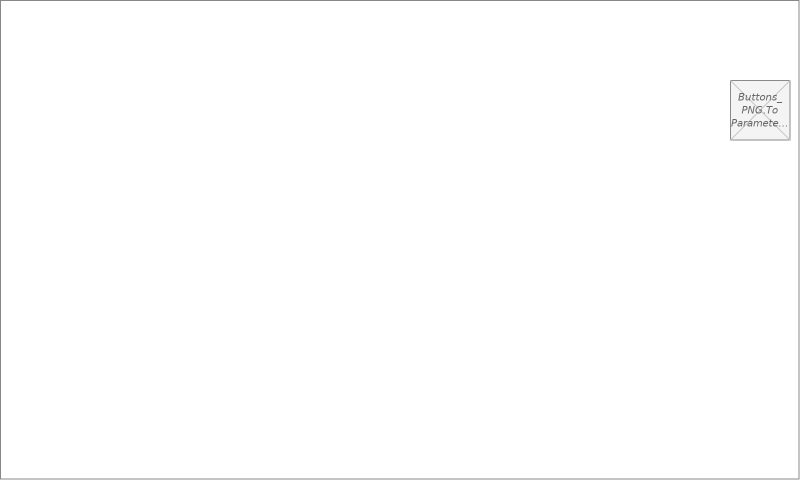
VISUALIZATION ParButton_PNG  // 800x480
VAR_IN_OUT
	bCmdParameter	: BOOL ; // to parameter screen
END_VAR
    Image (730,80 60x60), image: Buttons_PNG.To Parameter Screen
        OnMouseClick: toggle bCmdParameter
END_VISUALIZATION

(* stored: Version 1.1.0.1, ProductVersion 3.1.4024.11
   Visu ParButton_PNG: Id {9e342fb4-9cd9-4979-95df-eea2d44101f0} *)
